// TIA Portal V17 export
// export: Created 2025-03-20T13:42:40.4543954Z, ExportSetting WithDefaults, DisplayName Totally Integrated Automation Portal, DisplayVersion V17 Update 8, DisplayName TIA Portal Openness, DisplayVersion V17 Update 8, DisplayName TIA Portal Version Control Interface, DisplayVersion V17, DisplayName SINAMICS Startdrive Advanced, DisplayVersion V17 SP2, DisplayName SINAMICS Startdrive G110M, G120, G120C, G120D, G120P, G115D, DisplayVersion V17 SP2, DisplayName SINAMICS Startdrive G130, G150, S120, S150, SINAMICS MV, S210, DisplayVersion V17 SP2, DisplayName STEP 7 Professional, DisplayVersion V17 Update 8, DisplayName SINUMERIK ONE STEP 7 Toolbox, DisplayVersion V17 Update 12, DisplayName SINUMERIK 840D sl STEP 7 Toolbox, DisplayVersion V17 Update 12, DisplayName STEP 7 Safety, DisplayVersion V17 Update 6, DisplayName WinCC Advanced, DisplayVersion V17 Update 8
FUNCTION "FC22300_HOPPER_SYSTEM_ACTUATORS" : Void   // FC22300, LAD
TITLE = FC22300 HOPPER SYSTEM ACTUATORS
{ S7_Optimized_Access := 'TRUE' }
VERSION : 0.1
// stored: AutoNumber false, IsIECCheckEnabled false, SetENOAutomatically false, UDAEnableTagReadback false
BEGIN

REGION Network 1: //////////ACTUATORS HOPPERS UNIT 01//////////
END_REGION

REGION Network 2: CALL FB22301 TRANSFER POWDER VALVE HOPPER 1 UNIT 01
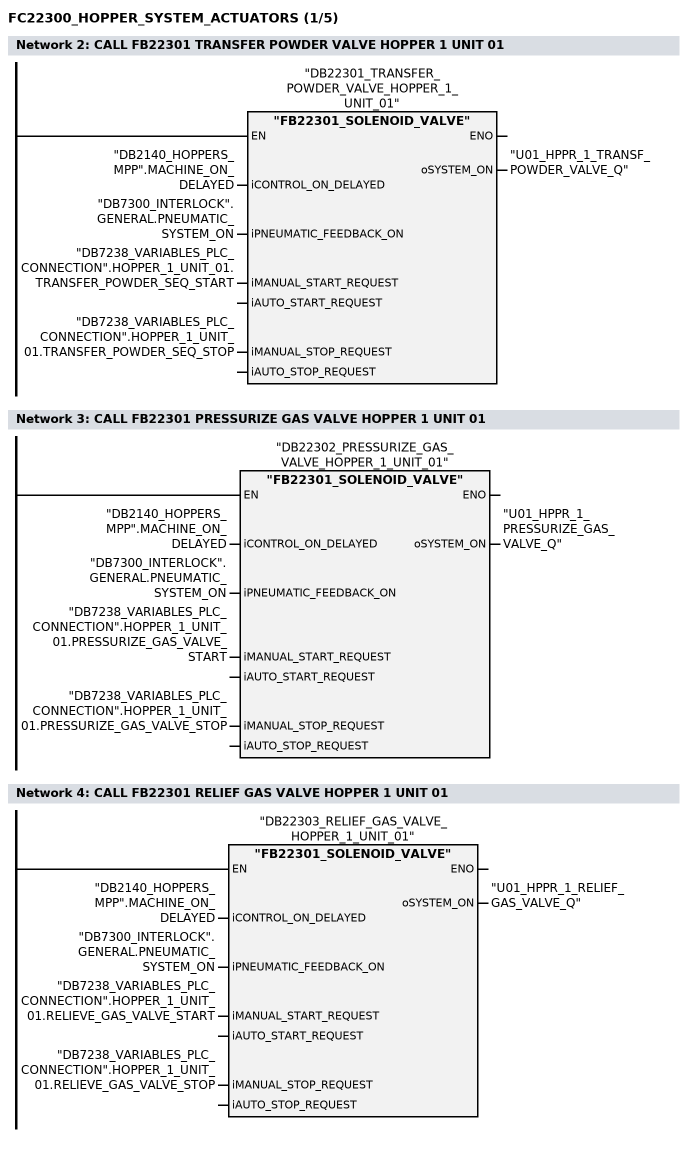
   RUNG wire#powerrail
      "DB22301_TRANSFER_POWDER_VALVE_HOPPER_1_UNIT_01"(iCONTROL_ON_DELAYED := "DB2140_HOPPERS_MPP".MACHINE_ON_DELAYED, iPNEUMATIC_FEEDBACK_ON := "DB7300_INTERLOCK".GENERAL.PNEUMATIC_SYSTEM_ON, iMANUAL_START_REQUEST := "DB7238_VARIABLES_PLC_CONNECTION".HOPPER_1_UNIT_01.TRANSFER_POWDER_SEQ_START, iAUTO_START_REQUEST :=, iMANUAL_STOP_REQUEST := "DB7238_VARIABLES_PLC_CONNECTION".HOPPER_1_UNIT_01.TRANSFER_POWDER_SEQ_STOP, iAUTO_STOP_REQUEST :=, oSYSTEM_ON => "U01_HPPR_1_TRANSF_POWDER_VALVE_Q")
   END_RUNG
   // the same network as SCL:
   "DB22301_TRANSFER_POWDER_VALVE_HOPPER_1_UNIT_01"(iCONTROL_ON_DELAYED := "DB2140_HOPPERS_MPP".MACHINE_ON_DELAYED,   // "FB22301_SOLENOID_VALVE"
                           iPNEUMATIC_FEEDBACK_ON := "DB7300_INTERLOCK".GENERAL.PNEUMATIC_SYSTEM_ON,
                           iMANUAL_START_REQUEST := "DB7238_VARIABLES_PLC_CONNECTION".HOPPER_1_UNIT_01.TRANSFER_POWDER_SEQ_START,
                           iMANUAL_STOP_REQUEST := "DB7238_VARIABLES_PLC_CONNECTION".HOPPER_1_UNIT_01.TRANSFER_POWDER_SEQ_STOP,
                           oSYSTEM_ON => "U01_HPPR_1_TRANSF_POWDER_VALVE_Q");
END_REGION

REGION Network 3: CALL FB22301 PRESSURIZE GAS VALVE HOPPER 1 UNIT 01
   RUNG wire#powerrail
      "DB22302_PRESSURIZE_GAS_VALVE_HOPPER_1_UNIT_01"(iCONTROL_ON_DELAYED := "DB2140_HOPPERS_MPP".MACHINE_ON_DELAYED, iPNEUMATIC_FEEDBACK_ON := "DB7300_INTERLOCK".GENERAL.PNEUMATIC_SYSTEM_ON, iMANUAL_START_REQUEST := "DB7238_VARIABLES_PLC_CONNECTION".HOPPER_1_UNIT_01.PRESSURIZE_GAS_VALVE_START, iAUTO_START_REQUEST :=, iMANUAL_STOP_REQUEST := "DB7238_VARIABLES_PLC_CONNECTION".HOPPER_1_UNIT_01.PRESSURIZE_GAS_VALVE_STOP, iAUTO_STOP_REQUEST :=, oSYSTEM_ON => "U01_HPPR_1_PRESSURIZE_GAS_VALVE_Q")
   END_RUNG
   // the same network as SCL:
   "DB22302_PRESSURIZE_GAS_VALVE_HOPPER_1_UNIT_01"(iCONTROL_ON_DELAYED := "DB2140_HOPPERS_MPP".MACHINE_ON_DELAYED,   // "FB22301_SOLENOID_VALVE"
                           iPNEUMATIC_FEEDBACK_ON := "DB7300_INTERLOCK".GENERAL.PNEUMATIC_SYSTEM_ON,
                           iMANUAL_START_REQUEST := "DB7238_VARIABLES_PLC_CONNECTION".HOPPER_1_UNIT_01.PRESSURIZE_GAS_VALVE_START,
                           iMANUAL_STOP_REQUEST := "DB7238_VARIABLES_PLC_CONNECTION".HOPPER_1_UNIT_01.PRESSURIZE_GAS_VALVE_STOP,
                           oSYSTEM_ON => "U01_HPPR_1_PRESSURIZE_GAS_VALVE_Q");
END_REGION

REGION Network 4: CALL FB22301 RELIEF GAS VALVE HOPPER 1 UNIT 01
   RUNG wire#powerrail
      "DB22303_RELIEF_GAS_VALVE_HOPPER_1_UNIT_01"(iCONTROL_ON_DELAYED := "DB2140_HOPPERS_MPP".MACHINE_ON_DELAYED, iPNEUMATIC_FEEDBACK_ON := "DB7300_INTERLOCK".GENERAL.PNEUMATIC_SYSTEM_ON, iMANUAL_START_REQUEST := "DB7238_VARIABLES_PLC_CONNECTION".HOPPER_1_UNIT_01.RELIEVE_GAS_VALVE_START, iAUTO_START_REQUEST :=, iMANUAL_STOP_REQUEST := "DB7238_VARIABLES_PLC_CONNECTION".HOPPER_1_UNIT_01.RELIEVE_GAS_VALVE_STOP, iAUTO_STOP_REQUEST :=, oSYSTEM_ON => "U01_HPPR_1_RELIEF_GAS_VALVE_Q")
   END_RUNG
   // the same network as SCL:
   "DB22303_RELIEF_GAS_VALVE_HOPPER_1_UNIT_01"(iCONTROL_ON_DELAYED := "DB2140_HOPPERS_MPP".MACHINE_ON_DELAYED,   // "FB22301_SOLENOID_VALVE"
                           iPNEUMATIC_FEEDBACK_ON := "DB7300_INTERLOCK".GENERAL.PNEUMATIC_SYSTEM_ON,
                           iMANUAL_START_REQUEST := "DB7238_VARIABLES_PLC_CONNECTION".HOPPER_1_UNIT_01.RELIEVE_GAS_VALVE_START,
                           iMANUAL_STOP_REQUEST := "DB7238_VARIABLES_PLC_CONNECTION".HOPPER_1_UNIT_01.RELIEVE_GAS_VALVE_STOP,
                           oSYSTEM_ON => "U01_HPPR_1_RELIEF_GAS_VALVE_Q");
END_REGION

REGION Network 5: CALL FB22301 TRANSFER POWDER VALVE HOPPER 2 UNIT 01
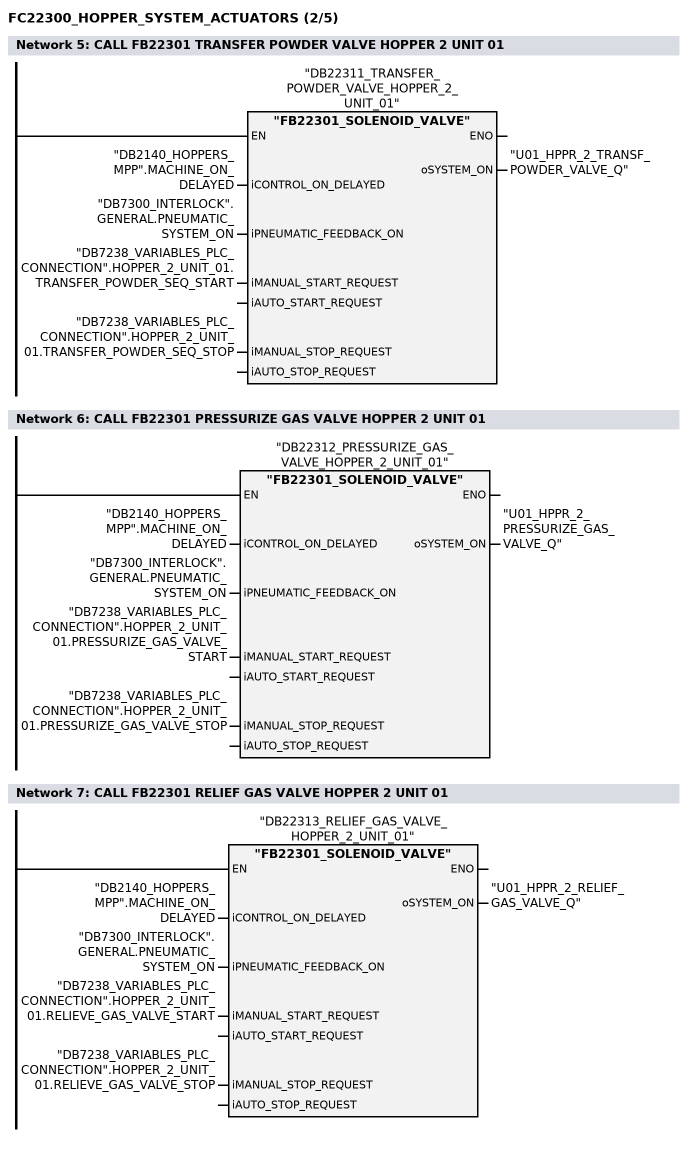
   RUNG wire#powerrail
      "DB22311_TRANSFER_POWDER_VALVE_HOPPER_2_UNIT_01"(iCONTROL_ON_DELAYED := "DB2140_HOPPERS_MPP".MACHINE_ON_DELAYED, iPNEUMATIC_FEEDBACK_ON := "DB7300_INTERLOCK".GENERAL.PNEUMATIC_SYSTEM_ON, iMANUAL_START_REQUEST := "DB7238_VARIABLES_PLC_CONNECTION".HOPPER_2_UNIT_01.TRANSFER_POWDER_SEQ_START, iAUTO_START_REQUEST :=, iMANUAL_STOP_REQUEST := "DB7238_VARIABLES_PLC_CONNECTION".HOPPER_2_UNIT_01.TRANSFER_POWDER_SEQ_STOP, iAUTO_STOP_REQUEST :=, oSYSTEM_ON => "U01_HPPR_2_TRANSF_POWDER_VALVE_Q")
   END_RUNG
   // the same network as SCL:
   "DB22311_TRANSFER_POWDER_VALVE_HOPPER_2_UNIT_01"(iCONTROL_ON_DELAYED := "DB2140_HOPPERS_MPP".MACHINE_ON_DELAYED,   // "FB22301_SOLENOID_VALVE"
                           iPNEUMATIC_FEEDBACK_ON := "DB7300_INTERLOCK".GENERAL.PNEUMATIC_SYSTEM_ON,
                           iMANUAL_START_REQUEST := "DB7238_VARIABLES_PLC_CONNECTION".HOPPER_2_UNIT_01.TRANSFER_POWDER_SEQ_START,
                           iMANUAL_STOP_REQUEST := "DB7238_VARIABLES_PLC_CONNECTION".HOPPER_2_UNIT_01.TRANSFER_POWDER_SEQ_STOP,
                           oSYSTEM_ON => "U01_HPPR_2_TRANSF_POWDER_VALVE_Q");
END_REGION

REGION Network 6: CALL FB22301 PRESSURIZE GAS VALVE HOPPER 2 UNIT 01
   RUNG wire#powerrail
      "DB22312_PRESSURIZE_GAS_VALVE_HOPPER_2_UNIT_01"(iCONTROL_ON_DELAYED := "DB2140_HOPPERS_MPP".MACHINE_ON_DELAYED, iPNEUMATIC_FEEDBACK_ON := "DB7300_INTERLOCK".GENERAL.PNEUMATIC_SYSTEM_ON, iMANUAL_START_REQUEST := "DB7238_VARIABLES_PLC_CONNECTION".HOPPER_2_UNIT_01.PRESSURIZE_GAS_VALVE_START, iAUTO_START_REQUEST :=, iMANUAL_STOP_REQUEST := "DB7238_VARIABLES_PLC_CONNECTION".HOPPER_2_UNIT_01.PRESSURIZE_GAS_VALVE_STOP, iAUTO_STOP_REQUEST :=, oSYSTEM_ON => "U01_HPPR_2_PRESSURIZE_GAS_VALVE_Q")
   END_RUNG
   // the same network as SCL:
   "DB22312_PRESSURIZE_GAS_VALVE_HOPPER_2_UNIT_01"(iCONTROL_ON_DELAYED := "DB2140_HOPPERS_MPP".MACHINE_ON_DELAYED,   // "FB22301_SOLENOID_VALVE"
                           iPNEUMATIC_FEEDBACK_ON := "DB7300_INTERLOCK".GENERAL.PNEUMATIC_SYSTEM_ON,
                           iMANUAL_START_REQUEST := "DB7238_VARIABLES_PLC_CONNECTION".HOPPER_2_UNIT_01.PRESSURIZE_GAS_VALVE_START,
                           iMANUAL_STOP_REQUEST := "DB7238_VARIABLES_PLC_CONNECTION".HOPPER_2_UNIT_01.PRESSURIZE_GAS_VALVE_STOP,
                           oSYSTEM_ON => "U01_HPPR_2_PRESSURIZE_GAS_VALVE_Q");
END_REGION

REGION Network 7: CALL FB22301 RELIEF GAS VALVE HOPPER 2 UNIT 01
   RUNG wire#powerrail
      "DB22313_RELIEF_GAS_VALVE_HOPPER_2_UNIT_01"(iCONTROL_ON_DELAYED := "DB2140_HOPPERS_MPP".MACHINE_ON_DELAYED, iPNEUMATIC_FEEDBACK_ON := "DB7300_INTERLOCK".GENERAL.PNEUMATIC_SYSTEM_ON, iMANUAL_START_REQUEST := "DB7238_VARIABLES_PLC_CONNECTION".HOPPER_2_UNIT_01.RELIEVE_GAS_VALVE_START, iAUTO_START_REQUEST :=, iMANUAL_STOP_REQUEST := "DB7238_VARIABLES_PLC_CONNECTION".HOPPER_2_UNIT_01.RELIEVE_GAS_VALVE_STOP, iAUTO_STOP_REQUEST :=, oSYSTEM_ON => "U01_HPPR_2_RELIEF_GAS_VALVE_Q")
   END_RUNG
   // the same network as SCL:
   "DB22313_RELIEF_GAS_VALVE_HOPPER_2_UNIT_01"(iCONTROL_ON_DELAYED := "DB2140_HOPPERS_MPP".MACHINE_ON_DELAYED,   // "FB22301_SOLENOID_VALVE"
                           iPNEUMATIC_FEEDBACK_ON := "DB7300_INTERLOCK".GENERAL.PNEUMATIC_SYSTEM_ON,
                           iMANUAL_START_REQUEST := "DB7238_VARIABLES_PLC_CONNECTION".HOPPER_2_UNIT_01.RELIEVE_GAS_VALVE_START,
                           iMANUAL_STOP_REQUEST := "DB7238_VARIABLES_PLC_CONNECTION".HOPPER_2_UNIT_01.RELIEVE_GAS_VALVE_STOP,
                           oSYSTEM_ON => "U01_HPPR_2_RELIEF_GAS_VALVE_Q");
END_REGION

REGION Network 8: //////////ACTUATORS HOPPERS UNIT 02//////////
END_REGION

REGION Network 9: CALL FB22301 TRANSFER POWDER VALVE HOPPER 1 UNIT 02
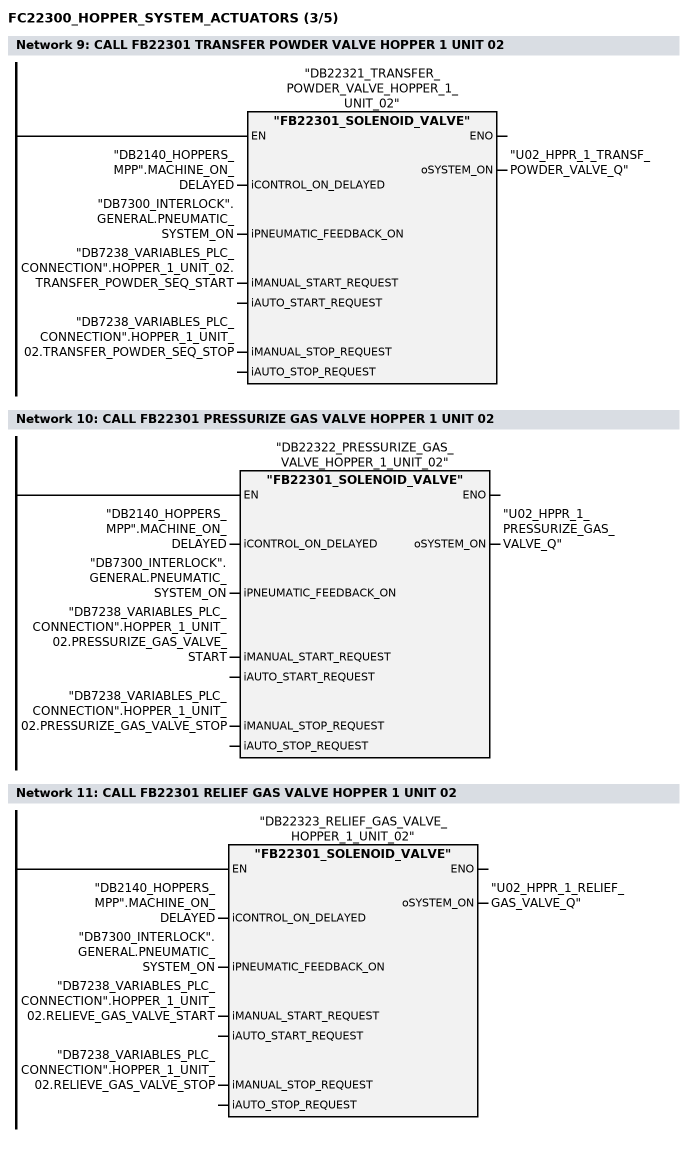
   RUNG wire#powerrail
      "DB22321_TRANSFER_POWDER_VALVE_HOPPER_1_UNIT_02"(iCONTROL_ON_DELAYED := "DB2140_HOPPERS_MPP".MACHINE_ON_DELAYED, iPNEUMATIC_FEEDBACK_ON := "DB7300_INTERLOCK".GENERAL.PNEUMATIC_SYSTEM_ON, iMANUAL_START_REQUEST := "DB7238_VARIABLES_PLC_CONNECTION".HOPPER_1_UNIT_02.TRANSFER_POWDER_SEQ_START, iAUTO_START_REQUEST :=, iMANUAL_STOP_REQUEST := "DB7238_VARIABLES_PLC_CONNECTION".HOPPER_1_UNIT_02.TRANSFER_POWDER_SEQ_STOP, iAUTO_STOP_REQUEST :=, oSYSTEM_ON => "U02_HPPR_1_TRANSF_POWDER_VALVE_Q")
   END_RUNG
   // the same network as SCL:
   "DB22321_TRANSFER_POWDER_VALVE_HOPPER_1_UNIT_02"(iCONTROL_ON_DELAYED := "DB2140_HOPPERS_MPP".MACHINE_ON_DELAYED,   // "FB22301_SOLENOID_VALVE"
                           iPNEUMATIC_FEEDBACK_ON := "DB7300_INTERLOCK".GENERAL.PNEUMATIC_SYSTEM_ON,
                           iMANUAL_START_REQUEST := "DB7238_VARIABLES_PLC_CONNECTION".HOPPER_1_UNIT_02.TRANSFER_POWDER_SEQ_START,
                           iMANUAL_STOP_REQUEST := "DB7238_VARIABLES_PLC_CONNECTION".HOPPER_1_UNIT_02.TRANSFER_POWDER_SEQ_STOP,
                           oSYSTEM_ON => "U02_HPPR_1_TRANSF_POWDER_VALVE_Q");
END_REGION

REGION Network 10: CALL FB22301 PRESSURIZE GAS VALVE HOPPER 1 UNIT 02
   RUNG wire#powerrail
      "DB22322_PRESSURIZE_GAS_VALVE_HOPPER_1_UNIT_02"(iCONTROL_ON_DELAYED := "DB2140_HOPPERS_MPP".MACHINE_ON_DELAYED, iPNEUMATIC_FEEDBACK_ON := "DB7300_INTERLOCK".GENERAL.PNEUMATIC_SYSTEM_ON, iMANUAL_START_REQUEST := "DB7238_VARIABLES_PLC_CONNECTION".HOPPER_1_UNIT_02.PRESSURIZE_GAS_VALVE_START, iAUTO_START_REQUEST :=, iMANUAL_STOP_REQUEST := "DB7238_VARIABLES_PLC_CONNECTION".HOPPER_1_UNIT_02.PRESSURIZE_GAS_VALVE_STOP, iAUTO_STOP_REQUEST :=, oSYSTEM_ON => "U02_HPPR_1_PRESSURIZE_GAS_VALVE_Q")
   END_RUNG
   // the same network as SCL:
   "DB22322_PRESSURIZE_GAS_VALVE_HOPPER_1_UNIT_02"(iCONTROL_ON_DELAYED := "DB2140_HOPPERS_MPP".MACHINE_ON_DELAYED,   // "FB22301_SOLENOID_VALVE"
                           iPNEUMATIC_FEEDBACK_ON := "DB7300_INTERLOCK".GENERAL.PNEUMATIC_SYSTEM_ON,
                           iMANUAL_START_REQUEST := "DB7238_VARIABLES_PLC_CONNECTION".HOPPER_1_UNIT_02.PRESSURIZE_GAS_VALVE_START,
                           iMANUAL_STOP_REQUEST := "DB7238_VARIABLES_PLC_CONNECTION".HOPPER_1_UNIT_02.PRESSURIZE_GAS_VALVE_STOP,
                           oSYSTEM_ON => "U02_HPPR_1_PRESSURIZE_GAS_VALVE_Q");
END_REGION

REGION Network 11: CALL FB22301 RELIEF GAS VALVE HOPPER 1 UNIT 02
   RUNG wire#powerrail
      "DB22323_RELIEF_GAS_VALVE_HOPPER_1_UNIT_02"(iCONTROL_ON_DELAYED := "DB2140_HOPPERS_MPP".MACHINE_ON_DELAYED, iPNEUMATIC_FEEDBACK_ON := "DB7300_INTERLOCK".GENERAL.PNEUMATIC_SYSTEM_ON, iMANUAL_START_REQUEST := "DB7238_VARIABLES_PLC_CONNECTION".HOPPER_1_UNIT_02.RELIEVE_GAS_VALVE_START, iAUTO_START_REQUEST :=, iMANUAL_STOP_REQUEST := "DB7238_VARIABLES_PLC_CONNECTION".HOPPER_1_UNIT_02.RELIEVE_GAS_VALVE_STOP, iAUTO_STOP_REQUEST :=, oSYSTEM_ON => "U02_HPPR_1_RELIEF_GAS_VALVE_Q")
   END_RUNG
   // the same network as SCL:
   "DB22323_RELIEF_GAS_VALVE_HOPPER_1_UNIT_02"(iCONTROL_ON_DELAYED := "DB2140_HOPPERS_MPP".MACHINE_ON_DELAYED,   // "FB22301_SOLENOID_VALVE"
                           iPNEUMATIC_FEEDBACK_ON := "DB7300_INTERLOCK".GENERAL.PNEUMATIC_SYSTEM_ON,
                           iMANUAL_START_REQUEST := "DB7238_VARIABLES_PLC_CONNECTION".HOPPER_1_UNIT_02.RELIEVE_GAS_VALVE_START,
                           iMANUAL_STOP_REQUEST := "DB7238_VARIABLES_PLC_CONNECTION".HOPPER_1_UNIT_02.RELIEVE_GAS_VALVE_STOP,
                           oSYSTEM_ON => "U02_HPPR_1_RELIEF_GAS_VALVE_Q");
END_REGION

REGION Network 12: CALL FB22301 TRANSFER POWDER VALVE HOPPER 2 UNIT 02
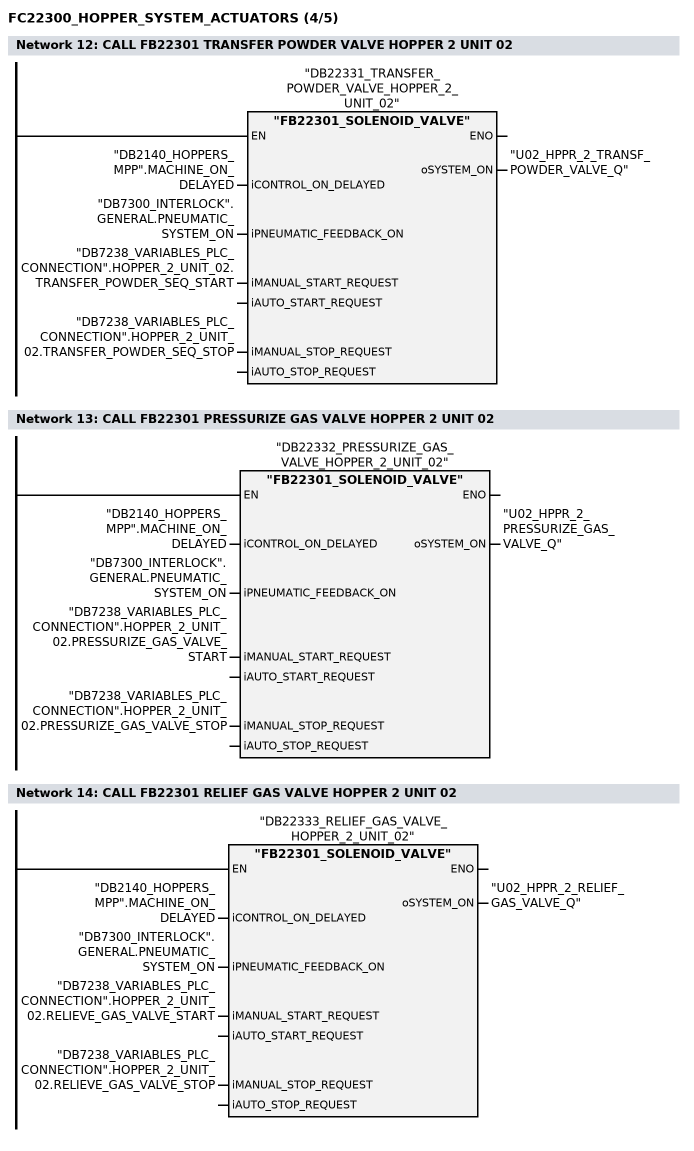
   RUNG wire#powerrail
      "DB22331_TRANSFER_POWDER_VALVE_HOPPER_2_UNIT_02"(iCONTROL_ON_DELAYED := "DB2140_HOPPERS_MPP".MACHINE_ON_DELAYED, iPNEUMATIC_FEEDBACK_ON := "DB7300_INTERLOCK".GENERAL.PNEUMATIC_SYSTEM_ON, iMANUAL_START_REQUEST := "DB7238_VARIABLES_PLC_CONNECTION".HOPPER_2_UNIT_02.TRANSFER_POWDER_SEQ_START, iAUTO_START_REQUEST :=, iMANUAL_STOP_REQUEST := "DB7238_VARIABLES_PLC_CONNECTION".HOPPER_2_UNIT_02.TRANSFER_POWDER_SEQ_STOP, iAUTO_STOP_REQUEST :=, oSYSTEM_ON => "U02_HPPR_2_TRANSF_POWDER_VALVE_Q")
   END_RUNG
   // the same network as SCL:
   "DB22331_TRANSFER_POWDER_VALVE_HOPPER_2_UNIT_02"(iCONTROL_ON_DELAYED := "DB2140_HOPPERS_MPP".MACHINE_ON_DELAYED,   // "FB22301_SOLENOID_VALVE"
                           iPNEUMATIC_FEEDBACK_ON := "DB7300_INTERLOCK".GENERAL.PNEUMATIC_SYSTEM_ON,
                           iMANUAL_START_REQUEST := "DB7238_VARIABLES_PLC_CONNECTION".HOPPER_2_UNIT_02.TRANSFER_POWDER_SEQ_START,
                           iMANUAL_STOP_REQUEST := "DB7238_VARIABLES_PLC_CONNECTION".HOPPER_2_UNIT_02.TRANSFER_POWDER_SEQ_STOP,
                           oSYSTEM_ON => "U02_HPPR_2_TRANSF_POWDER_VALVE_Q");
END_REGION

REGION Network 13: CALL FB22301 PRESSURIZE GAS VALVE HOPPER 2 UNIT 02
   RUNG wire#powerrail
      "DB22332_PRESSURIZE_GAS_VALVE_HOPPER_2_UNIT_02"(iCONTROL_ON_DELAYED := "DB2140_HOPPERS_MPP".MACHINE_ON_DELAYED, iPNEUMATIC_FEEDBACK_ON := "DB7300_INTERLOCK".GENERAL.PNEUMATIC_SYSTEM_ON, iMANUAL_START_REQUEST := "DB7238_VARIABLES_PLC_CONNECTION".HOPPER_2_UNIT_02.PRESSURIZE_GAS_VALVE_START, iAUTO_START_REQUEST :=, iMANUAL_STOP_REQUEST := "DB7238_VARIABLES_PLC_CONNECTION".HOPPER_2_UNIT_02.PRESSURIZE_GAS_VALVE_STOP, iAUTO_STOP_REQUEST :=, oSYSTEM_ON => "U02_HPPR_2_PRESSURIZE_GAS_VALVE_Q")
   END_RUNG
   // the same network as SCL:
   "DB22332_PRESSURIZE_GAS_VALVE_HOPPER_2_UNIT_02"(iCONTROL_ON_DELAYED := "DB2140_HOPPERS_MPP".MACHINE_ON_DELAYED,   // "FB22301_SOLENOID_VALVE"
                           iPNEUMATIC_FEEDBACK_ON := "DB7300_INTERLOCK".GENERAL.PNEUMATIC_SYSTEM_ON,
                           iMANUAL_START_REQUEST := "DB7238_VARIABLES_PLC_CONNECTION".HOPPER_2_UNIT_02.PRESSURIZE_GAS_VALVE_START,
                           iMANUAL_STOP_REQUEST := "DB7238_VARIABLES_PLC_CONNECTION".HOPPER_2_UNIT_02.PRESSURIZE_GAS_VALVE_STOP,
                           oSYSTEM_ON => "U02_HPPR_2_PRESSURIZE_GAS_VALVE_Q");
END_REGION

REGION Network 14: CALL FB22301 RELIEF GAS VALVE HOPPER 2 UNIT 02
   RUNG wire#powerrail
      "DB22333_RELIEF_GAS_VALVE_HOPPER_2_UNIT_02"(iCONTROL_ON_DELAYED := "DB2140_HOPPERS_MPP".MACHINE_ON_DELAYED, iPNEUMATIC_FEEDBACK_ON := "DB7300_INTERLOCK".GENERAL.PNEUMATIC_SYSTEM_ON, iMANUAL_START_REQUEST := "DB7238_VARIABLES_PLC_CONNECTION".HOPPER_2_UNIT_02.RELIEVE_GAS_VALVE_START, iAUTO_START_REQUEST :=, iMANUAL_STOP_REQUEST := "DB7238_VARIABLES_PLC_CONNECTION".HOPPER_2_UNIT_02.RELIEVE_GAS_VALVE_STOP, iAUTO_STOP_REQUEST :=, oSYSTEM_ON => "U02_HPPR_2_RELIEF_GAS_VALVE_Q")
   END_RUNG
   // the same network as SCL:
   "DB22333_RELIEF_GAS_VALVE_HOPPER_2_UNIT_02"(iCONTROL_ON_DELAYED := "DB2140_HOPPERS_MPP".MACHINE_ON_DELAYED,   // "FB22301_SOLENOID_VALVE"
                           iPNEUMATIC_FEEDBACK_ON := "DB7300_INTERLOCK".GENERAL.PNEUMATIC_SYSTEM_ON,
                           iMANUAL_START_REQUEST := "DB7238_VARIABLES_PLC_CONNECTION".HOPPER_2_UNIT_02.RELIEVE_GAS_VALVE_START,
                           iMANUAL_STOP_REQUEST := "DB7238_VARIABLES_PLC_CONNECTION".HOPPER_2_UNIT_02.RELIEVE_GAS_VALVE_STOP,
                           oSYSTEM_ON => "U02_HPPR_2_RELIEF_GAS_VALVE_Q");
END_REGION

REGION Network 15: CALL FB22301 TRANSFER POWDER VALVE HOPPER 3 UNIT 02
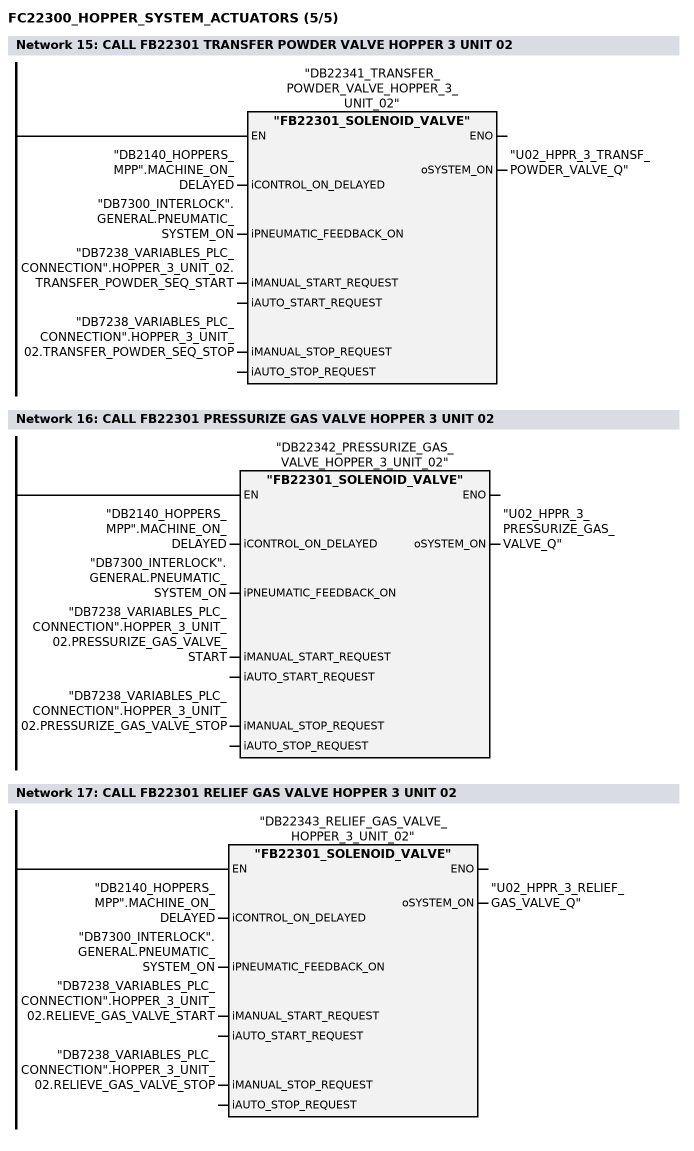
   RUNG wire#powerrail
      "DB22341_TRANSFER_POWDER_VALVE_HOPPER_3_UNIT_02"(iCONTROL_ON_DELAYED := "DB2140_HOPPERS_MPP".MACHINE_ON_DELAYED, iPNEUMATIC_FEEDBACK_ON := "DB7300_INTERLOCK".GENERAL.PNEUMATIC_SYSTEM_ON, iMANUAL_START_REQUEST := "DB7238_VARIABLES_PLC_CONNECTION".HOPPER_3_UNIT_02.TRANSFER_POWDER_SEQ_START, iAUTO_START_REQUEST :=, iMANUAL_STOP_REQUEST := "DB7238_VARIABLES_PLC_CONNECTION".HOPPER_3_UNIT_02.TRANSFER_POWDER_SEQ_STOP, iAUTO_STOP_REQUEST :=, oSYSTEM_ON => "U02_HPPR_3_TRANSF_POWDER_VALVE_Q")
   END_RUNG
   // the same network as SCL:
   "DB22341_TRANSFER_POWDER_VALVE_HOPPER_3_UNIT_02"(iCONTROL_ON_DELAYED := "DB2140_HOPPERS_MPP".MACHINE_ON_DELAYED,   // "FB22301_SOLENOID_VALVE"
                           iPNEUMATIC_FEEDBACK_ON := "DB7300_INTERLOCK".GENERAL.PNEUMATIC_SYSTEM_ON,
                           iMANUAL_START_REQUEST := "DB7238_VARIABLES_PLC_CONNECTION".HOPPER_3_UNIT_02.TRANSFER_POWDER_SEQ_START,
                           iMANUAL_STOP_REQUEST := "DB7238_VARIABLES_PLC_CONNECTION".HOPPER_3_UNIT_02.TRANSFER_POWDER_SEQ_STOP,
                           oSYSTEM_ON => "U02_HPPR_3_TRANSF_POWDER_VALVE_Q");
END_REGION

REGION Network 16: CALL FB22301 PRESSURIZE GAS VALVE HOPPER 3 UNIT 02
   RUNG wire#powerrail
      "DB22342_PRESSURIZE_GAS_VALVE_HOPPER_3_UNIT_02"(iCONTROL_ON_DELAYED := "DB2140_HOPPERS_MPP".MACHINE_ON_DELAYED, iPNEUMATIC_FEEDBACK_ON := "DB7300_INTERLOCK".GENERAL.PNEUMATIC_SYSTEM_ON, iMANUAL_START_REQUEST := "DB7238_VARIABLES_PLC_CONNECTION".HOPPER_3_UNIT_02.PRESSURIZE_GAS_VALVE_START, iAUTO_START_REQUEST :=, iMANUAL_STOP_REQUEST := "DB7238_VARIABLES_PLC_CONNECTION".HOPPER_3_UNIT_02.PRESSURIZE_GAS_VALVE_STOP, iAUTO_STOP_REQUEST :=, oSYSTEM_ON => "U02_HPPR_3_PRESSURIZE_GAS_VALVE_Q")
   END_RUNG
   // the same network as SCL:
   "DB22342_PRESSURIZE_GAS_VALVE_HOPPER_3_UNIT_02"(iCONTROL_ON_DELAYED := "DB2140_HOPPERS_MPP".MACHINE_ON_DELAYED,   // "FB22301_SOLENOID_VALVE"
                           iPNEUMATIC_FEEDBACK_ON := "DB7300_INTERLOCK".GENERAL.PNEUMATIC_SYSTEM_ON,
                           iMANUAL_START_REQUEST := "DB7238_VARIABLES_PLC_CONNECTION".HOPPER_3_UNIT_02.PRESSURIZE_GAS_VALVE_START,
                           iMANUAL_STOP_REQUEST := "DB7238_VARIABLES_PLC_CONNECTION".HOPPER_3_UNIT_02.PRESSURIZE_GAS_VALVE_STOP,
                           oSYSTEM_ON => "U02_HPPR_3_PRESSURIZE_GAS_VALVE_Q");
END_REGION

REGION Network 17: CALL FB22301 RELIEF GAS VALVE HOPPER 3 UNIT 02
   RUNG wire#powerrail
      "DB22343_RELIEF_GAS_VALVE_HOPPER_3_UNIT_02"(iCONTROL_ON_DELAYED := "DB2140_HOPPERS_MPP".MACHINE_ON_DELAYED, iPNEUMATIC_FEEDBACK_ON := "DB7300_INTERLOCK".GENERAL.PNEUMATIC_SYSTEM_ON, iMANUAL_START_REQUEST := "DB7238_VARIABLES_PLC_CONNECTION".HOPPER_3_UNIT_02.RELIEVE_GAS_VALVE_START, iAUTO_START_REQUEST :=, iMANUAL_STOP_REQUEST := "DB7238_VARIABLES_PLC_CONNECTION".HOPPER_3_UNIT_02.RELIEVE_GAS_VALVE_STOP, iAUTO_STOP_REQUEST :=, oSYSTEM_ON => "U02_HPPR_3_RELIEF_GAS_VALVE_Q")
   END_RUNG
   // the same network as SCL:
   "DB22343_RELIEF_GAS_VALVE_HOPPER_3_UNIT_02"(iCONTROL_ON_DELAYED := "DB2140_HOPPERS_MPP".MACHINE_ON_DELAYED,   // "FB22301_SOLENOID_VALVE"
                           iPNEUMATIC_FEEDBACK_ON := "DB7300_INTERLOCK".GENERAL.PNEUMATIC_SYSTEM_ON,
                           iMANUAL_START_REQUEST := "DB7238_VARIABLES_PLC_CONNECTION".HOPPER_3_UNIT_02.RELIEVE_GAS_VALVE_START,
                           iMANUAL_STOP_REQUEST := "DB7238_VARIABLES_PLC_CONNECTION".HOPPER_3_UNIT_02.RELIEVE_GAS_VALVE_STOP,
                           oSYSTEM_ON => "U02_HPPR_3_RELIEF_GAS_VALVE_Q");
END_REGION
END_FUNCTION
